FUNCTION F_GetCommandValue : POINTER TO FB_LinearActuator
VAR_INPUT
    nX : INT;
    sY : STRING;
END_VAR
VAR
    i : INT;
    pResult: POINTER TO FB_LinearActuator;
END_VAR

FOR i := 1 TO nEntryCount DO
    IF aLookupTable[i].nX = nX AND aLookupTable[i].sY = sY THEN
			pResult := aLookupTable[i].sValue;
        EXIT;
    END_IF;
END_FOR;

F_GetCommandValue := pResult;

END_FUNCTION

(* stored: Version 1.1.0.1, ProductVersion 3.1.4026.11
   POU F_GetCommandValue: Id {de4afad7-ea2b-4397-ab7f-0f6497443525}, SpecialFunc None *)
